// TIA Portal V19 export
TYPE "Positioning_MOL_Machine_Alr"
// stored: Access Published
   STRUCT
      Ax_NotHomed : Bool;   // Axis is NOT homed / refereced
      Ax : "OOAx_Alr";   // ON-OFF AXIS
      Motor : "MotorSAlr";   // MOTOR
   END_STRUCT;
END_TYPE
